{attribute 'GeneratedUsingTerminal: EL3174-0002-0017'}
{attribute addProperty VendorId "#x00000002"}
{attribute addProperty BoxType "EL3174-0002-0017"}
{attribute addProperty Description "EL3174-0002 4Ch. Ana. Input +/-10V, +/-20mA 16 Bit, Isolated Channels"}
{attribute addProperty Physics "KK"}
{attribute addProperty Id "AI_Standard_Channel_1AT %I*AI_Standard_Channel_A8DF64E310AI_Standard_Channel_2AT %I*AI_Standard_Channel_A8DF64E310AI_Standard_Channel_3AT %I*AI_Standard_Channel_A8DF64E310AI_Standard_Channel_4AT %I*AI_Standard_Channel_A8DF64E310WcStateAT %I*WcState_9091E0EB2InfoDataAT %I*InfoData_23CBA8372"}
{attribute addProperty CRC "3072065346"}
{attribute addProperty Size "44"}
TYPE EL3174_B71BFF42 EXTENDS TcoIo.EtcSlaveTerminalBase_947E5A46 :
STRUCT
    {attribute addProperty Name "AI_Standard_Channel_1"}
    AI_Standard_Channel_1 : AI_Standard_Channel_A8DF64E3;
    {attribute addProperty Name "AI_Standard_Channel_2"}
    AI_Standard_Channel_2 : AI_Standard_Channel_A8DF64E3;
    {attribute addProperty Name "AI_Standard_Channel_3"}
    AI_Standard_Channel_3 : AI_Standard_Channel_A8DF64E3;
    {attribute addProperty Name "AI_Standard_Channel_4"}
    AI_Standard_Channel_4 : AI_Standard_Channel_A8DF64E3;
    {attribute addProperty Name "WcState"}
    WcState : TcoIo.WcState_9091E0EB;
    {attribute addProperty Name "InfoData"}
    InfoData : TcoIo.InfoData_23CBA837;
END_STRUCT
END_TYPE

(* stored: Version 1.2.0.0, ProductVersion 3.1.4024.11
   DUT EL3174_B71BFF42: Id {acefba29-5d04-0950-0b7a-e38be1809c5e} *)
